TYPE ANA_Standard :
STRUCT
	
	MesData		: ANA; (* (NA) Child struct *)
END_STRUCT
END_TYPE

(* stored: Version 1.1.0.1, ProductVersion 3.1.4024.13
   DUT ANA_Standard: Id {aa338462-e780-411b-9426-b27ce6a5bf67} *)
